Yaskawa INFORM job: long_pipe_cylinder_program.JBI

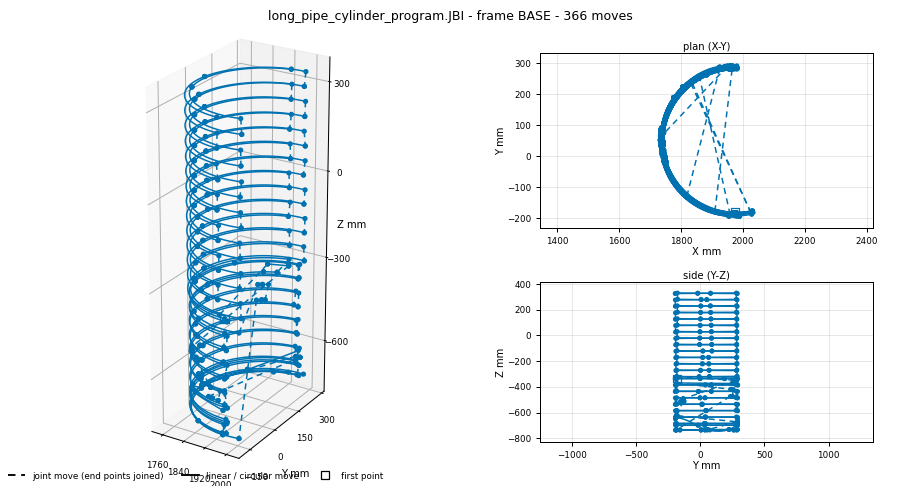
[picture p0: tool path of long_pipe_cylinder_program.JBI in frame BASE, 366 of 497 moves have a stored position in this frame; points joined in program order, loops and branches not executed]
/JOB
//NAME long_pipe_cylinder_program
//POS
///NPOS 488,0,488,0,0,0
///TOOL 0
///POSTYPE BASE
///RECTAN
///RCONF 0,0,0,0,0,0,0,0,0,0,0,0,0,0,0,0,0,0,0,0,0,0,0,0
C00000=1972.508334,-180.722400,-334.797447,175.000000,-89.735184,90.500621
C00001=1972.508334,-180.722400,-334.797447,175.000000,-89.735184,90.500621
C00002=1736.408412,94.560328,-335.864178,175.000000,-89.992940,-9.264169
C00003=1775.133773,190.860038,-336.344108,-5.000000,-89.891094,145.451183
C00004=1775.133773,190.860038,-336.344108,-5.000000,-89.891094,145.451183
C00005=1775.133773,190.860038,-336.344108,-5.000000,-89.891094,145.451183
C00006=1827.250532,245.393825,-336.642454,5.000000,-89.819004,127.146501
C00007=1960.064613,293.278571,-336.981034,-5.000000,-89.737192,92.507006
C00008=1958.169423,292.965805,-385.452719,-5.000000,-89.737685,92.955150
C00009=1958.169423,292.965805,-385.452719,-5.000000,-89.737685,92.955150
C00010=1816.172076,236.277891,-385.065300,-5.000000,-89.831298,130.571443
C00011=1735.474228,88.397981,-384.309626,-175.000000,-89.986107,-7.813258
C00012=1735.474228,88.397981,-384.309626,-175.000000,-89.986107,-7.813258
C00013=1735.474228,88.397981,-384.309626,-175.000000,-89.986107,-7.813258
C00014=1785.900263,-92.792903,-383.515122,175.000000,-89.794130,38.916534
C00015=1972.374520,-180.947584,-383.271088,175.000000,-89.735163,90.478593
C00016=1969.015250,-181.182972,-433.141929,175.000000,-89.734453,89.677478
C00017=1969.015250,-181.182972,-433.141929,175.000000,-89.734453,89.677478
C00018=1788.215870,-95.899703,-433.377664,175.000000,-89.791415,39.815407
C00019=1735.352609,87.595450,-434.180691,175.000000,-89.985451,-7.673859
C00020=1735.352609,87.595450,-434.180691,175.000000,-89.985451,-7.673859
C00021=1735.352609,87.595450,-434.180691,175.000000,-89.985451,-7.673859
C00022=1805.125009,226.010115,-434.882928,-5.000000,-89.844866,134.170721
C00023=1947.373302,291.934457,-435.313330,5.000000,-89.740867,95.560664
C00024=1940.676594,290.957693,-485.903239,5.000000,-89.743112,97.178090
C00025=1940.676594,290.957693,-485.903239,5.000000,-89.743112,97.178090
C00026=1806.475544,227.120060,-485.489579,5.000000,-89.843066,133.702612
C00027=1733.832144,38.186072,-484.550920,-175.000000,-89.930125,5.000000
C00028=1733.832144,38.186072,-484.550920,-175.000000,-89.930125,5.000000
C00029=1733.832144,38.186072,-484.550920,-175.000000,-89.930125,5.000000
C00030=1801.988125,-111.319855,-483.918715,175.000000,-89.777364,44.777879
C00031=1967.484314,-181.404185,-483.739882,-175.000000,-89.734152,89.318297
C00032=1979.401274,-181.476259,-533.747056,175.000000,-89.736874,92.209028
C00033=1979.401274,-181.476259,-533.747056,175.000000,-89.736874,92.209028
C00034=1821.064603,-128.831806,-533.851447,175.000000,-89.762098,51.008369
C00035=1736.221976,17.364408,-534.453644,175.000000,-89.907608,9.246629
C00036=1736.221976,17.364408,-534.453644,175.000000,-89.907608,9.246629
C00037=1736.221976,17.364408,-534.453644,175.000000,-89.907608,9.246629
C00038=1787.842464,206.956552,-535.376849,5.000000,-89.869317,140.291943
C00039=1956.911466,292.208440,-535.920338,5.000000,-89.737992,93.227517
C00040=1950.680326,291.548047,-585.654124,5.000000,-89.739789,94.726243
C00041=1950.680326,291.548047,-585.654124,5.000000,-89.739789,94.726243
C00042=1792.775612,212.526390,-585.149306,5.000000,-89.861770,138.445142
C00043=1733.319404,44.964590,-584.321201,175.000000,-89.938134,5.000000
C00044=1733.319404,44.964590,-584.321201,175.000000,-89.938134,5.000000
C00045=1733.319404,44.964590,-584.321201,175.000000,-89.938134,5.000000
C00046=1826.635210,-133.468869,-583.577209,-175.000000,-89.758362,52.733042
C00047=1971.739744,-181.877826,-583.480783,175.000000,-89.735062,90.367778
C00048=1971.702534,-182.110717,-633.797386,-175.000000,-89.735064,90.369485
C00049=1971.702534,-182.110717,-633.797386,-175.000000,-89.735064,90.369485
C00050=1827.055515,-134.054392,-633.892582,175.000000,-89.758066,52.873969
C00051=1733.473975,40.872659,-634.620107,175.000000,-89.933859,5.000000
C00052=1733.473975,40.872659,-634.620107,175.000000,-89.933859,5.000000
C00053=1733.473975,40.872659,-634.620107,175.000000,-89.933859,5.000000
C00054=1792.290752,211.795028,-635.463207,-5.000000,-89.862421,138.605884
C00055=1947.450954,291.030161,-635.966599,5.000000,-89.740785,95.498948
C00056=1950.402769,291.069729,-685.572290,5.000000,-89.739847,94.772222
C00057=1950.402769,291.069729,-685.572290,5.000000,-89.739847,94.772222
C00058=1804.325673,224.287077,-685.134545,5.000000,-89.845621,134.366136
C00059=1733.942614,33.751843,-684.190461,175.000000,-89.926259,5.086090
C00060=1733.942614,33.751843,-684.190461,175.000000,-89.926259,5.086090
C00061=1733.942614,33.751843,-684.190461,175.000000,-89.926259,5.086090
C00062=1831.125071,-137.328437,-683.483916,175.000000,-89.755535,54.110506
C00063=1976.553212,-182.258277,-683.403882,-175.000000,-89.736196,91.552306
C00064=1977.797365,-182.451641,-733.470089,-175.000000,-89.736513,91.863719
C00065=1977.797365,-182.451641,-733.470089,-175.000000,-89.736513,91.863719
C00066=1832.240189,-138.393667,-733.545972,-175.000000,-89.754849,54.455487
C00067=1732.965067,54.885977,-734.353455,175.000000,-89.949963,-5.000000
C00068=1732.965067,54.885977,-734.353455,175.000000,-89.949963,-5.000000
C00069=1732.965067,54.885977,-734.353455,175.000000,-89.949963,-5.000000
C00070=1795.566929,215.069330,-735.150167,5.000000,-89.857527,137.391169
C00071=1959.659103,291.432152,-648.357585,-5.000000,-89.737207,92.520217
C00072=1954.235485,290.902862,-698.306483,-5.000000,-89.738684,93.822137
C00073=1954.235485,290.902862,-698.306483,-5.000000,-89.738684,93.822137
C00074=1797.089158,216.524941,-698.129153,-5.000000,-89.855307,136.834972
C00075=1743.660264,-16.242507,-697.715930,175.000000,-89.872933,17.309849
C00076=1743.660264,-16.242507,-697.715930,175.000000,-89.872933,17.309849
C00077=1743.660264,-16.242507,-697.715930,175.000000,-89.872933,17.309849
C00078=1826.609334,-134.510209,-697.541573,175.000000,-89.758266,52.778835
C00079=1980.284076,-182.588600,-697.509479,175.000000,-89.737158,92.475638
C00080=1963.195867,-182.887095,-735.326535,-175.000000,-89.733394,88.353627
C00081=1963.195867,-182.887095,-735.326535,-175.000000,-89.733394,88.353627
C00082=1816.510486,-126.597836,-735.374855,175.000000,-89.765173,49.658472
C00083=1737.516210,7.512714,-735.577440,-175.000000,-89.898405,11.339291
C00084=1737.516210,7.512714,-735.577440,-175.000000,-89.898405,11.339291
C00085=1737.516210,7.512714,-735.577440,-175.000000,-89.898405,11.339291
C00086=1770.184921,181.794183,-735.884464,5.000000,-89.899679,147.427154
C00087=1925.404749,287.022342,-736.113649,-175.000000,-60.000000,-79.157724
C00088=1954.714747,-193.319715,326.566406,5.000000,-89.456000,-93.567339
C00089=1954.714747,-193.319715,326.566406,5.000000,-89.456000,-93.567339
C00090=1779.619946,-99.163395,327.312391,-5.000000,-89.635698,-142.973579
C00091=1734.628999,81.575451,328.985260,175.000000,-89.961340,-9.072278
C00092=1734.628999,81.575451,328.985260,175.000000,-89.961340,-9.072278
C00093=1734.628999,81.575451,328.985260,175.000000,-89.961340,-9.072278
C00094=1817.345576,226.880631,330.428549,-175.000000,-89.613678,-50.226634
C00095=1980.685637,281.657087,331.081997,-175.000000,-89.456271,-92.692092
C00096=1975.331224,282.321864,281.169566,-175.000000,-89.456908,-91.391494
C00097=1975.331224,282.321864,281.169566,-175.000000,-89.456908,-91.391494
C00098=1806.653771,217.858300,280.420044,175.000000,-89.637458,-46.774255
C00099=1731.827481,52.492803,278.793480,5.000000,-89.970734,175.000000
C00100=1731.827481,52.492803,278.793480,5.000000,-89.970734,175.000000
C00101=1731.827481,52.492803,278.793480,5.000000,-89.970734,175.000000
C00102=1788.634891,-109.869774,277.304259,5.000000,-89.612008,-139.519963
C00103=1955.354656,-192.883892,276.656769,5.000000,-89.456036,-93.422839
C00104=1953.241860,-192.282365,227.745608,5.000000,-89.455922,-93.942585
C00105=1953.241860,-192.282365,227.745608,5.000000,-89.455922,-93.942585
C00106=1805.749479,-127.416353,228.237298,5.000000,-89.574365,-133.539245
C00107=1734.368459,80.302128,230.143603,175.000000,-89.966442,-8.533915
C00108=1734.368459,80.302128,230.143603,175.000000,-89.966442,-8.533915
C00109=1734.368459,80.302128,230.143603,175.000000,-89.966442,-8.533915
C00110=1827.599341,235.823990,231.692259,175.000000,-89.593399,-53.345559
C00111=1980.201861,282.618326,232.261298,-175.000000,-89.456324,-92.555776
C00112=1977.844791,283.196392,181.219557,175.000000,-89.456586,-91.977383
C00113=1977.844791,283.196392,181.219557,175.000000,-89.456586,-91.977383
C00114=1800.614926,212.840705,180.407208,175.000000,-89.652270,-44.715535
C00115=1734.671921,82.485007,179.119248,175.000000,-89.962516,-8.948170
C00116=1734.671921,82.485007,179.119248,175.000000,-89.962516,-8.948170
C00117=1734.671921,82.485007,179.119248,175.000000,-89.962516,-8.948170
C00118=1775.815306,-92.383268,177.498740,5.000000,-89.647135,-144.574723
C00119=1951.488512,-191.668695,176.704704,-5.000000,-89.455862,-94.376235
C00120=1956.296565,-191.511118,126.598565,5.000000,-89.456090,-93.225427
C00121=1956.296565,-191.511118,126.598565,5.000000,-89.456090,-93.225427
C00122=1767.398896,-79.172346,127.505165,5.000000,-89.674478,-148.258247
C00123=1734.897298,84.109732,129.023199,175.000000,-89.959857,-9.228817
C00124=1734.897298,84.109732,129.023199,175.000000,-89.959857,-9.228817
C00125=1734.897298,84.109732,129.023199,175.000000,-89.959857,-9.228817
C00126=1813.190108,225.089245,130.421898,-175.000000,-89.622936,-48.858885
C00127=1976.049655,283.726966,131.111484,175.000000,-89.456824,-91.534787
C00128=1980.343703,284.039913,81.981880,175.000000,-89.456323,-92.560087
C00129=1980.343703,284.039913,81.981880,175.000000,-89.456323,-92.560087
C00130=1804.393738,217.432812,81.206058,-175.000000,-89.643208,-45.967475
C00131=1735.189988,86.095506,79.906112,-175.000000,-89.956341,-9.600136
C00132=1735.189988,86.095506,79.906112,-175.000000,-89.956341,-9.600136
C00133=1735.189988,86.095506,79.906112,-175.000000,-89.956341,-9.600136
C00134=1760.047671,-65.884409,78.488690,5.000000,-89.702230,-151.824094
C00135=1954.293720,-190.922109,77.466362,5.000000,-89.455966,-93.718563
C00136=1952.261030,-190.301711,27.124546,5.000000,-89.455880,-94.219424
C00137=1952.261030,-190.301711,27.124546,5.000000,-89.455880,-94.219424
C00138=1771.749852,-84.881332,27.972626,-5.000000,-89.660171,-146.354530
C00139=1735.436141,87.763326,29.576092,175.000000,-89.953585,-9.891308
C00140=1735.436141,87.763326,29.576092,175.000000,-89.953585,-9.891308
C00141=1735.436141,87.763326,29.576092,175.000000,-89.953585,-9.891308
C00142=1807.857666,221.152725,30.898117,175.000000,-89.635134,-47.103300
C00143=1980.425383,284.514593,31.640434,175.000000,-89.456319,-92.569770
C00144=1974.499385,285.179775,-18.267395,-175.000000,-89.457069,-91.131550
C00145=1974.499385,285.179775,-18.267395,-175.000000,-89.457069,-91.131550
C00146=1792.515923,205.949239,-19.167650,175.000000,-89.673928,-41.810930
C00147=1735.592913,88.893179,-20.322308,175.000000,-89.952063,-10.052118
C00148=1735.592913,88.893179,-20.322308,175.000000,-89.952063,-10.052118
C00149=1735.592913,88.893179,-20.322308,175.000000,-89.952063,-10.052118
C00150=1768.035641,-78.584750,-21.880090,-5.000000,-89.672697,-148.023907
C00151=1957.112660,-190.135299,-22.779084,-5.000000,-89.456142,-93.058269
C00152=1954.940310,-189.534063,-72.713074,-5.000000,-89.455994,-93.592390
C00153=1954.940310,-189.534063,-72.713074,-5.000000,-89.455994,-93.592390
C00154=1772.096519,-84.332612,-71.868996,5.000000,-89.659321,-146.239795
C00155=1735.849108,90.560889,-70.244197,-175.000000,-89.949296,-10.344614
C00156=1735.849108,90.560889,-70.244197,-175.000000,-89.949296,-10.344614
C00157=1735.849108,90.560889,-70.244197,-175.000000,-89.949296,-10.344614
C00158=1807.335261,221.533864,-68.945810,175.000000,-89.636539,-46.904132
C00159=1980.981190,285.437832,-68.197471,-175.000000,-89.456274,-92.683940
C00160=1976.954500,286.068414,-118.357107,175.000000,-89.456730,-91.703253
C00161=1976.954500,286.068414,-118.357107,175.000000,-89.456730,-91.703253
C00162=1794.437453,208.928718,-119.238021,175.000000,-89.668930,-42.471118
C00163=1736.086800,92.097439,-120.391733,-175.000000,-89.946837,-10.604717
C00164=1736.086800,92.097439,-120.391733,-175.000000,-89.946837,-10.604717
C00165=1736.086800,92.097439,-120.391733,-175.000000,-89.946837,-10.604717
C00166=1770.555957,-81.460267,-122.005364,-5.000000,-89.664470,-146.931728
C00167=1957.534905,-189.205848,-122.870092,-5.000000,-89.456169,-92.976329
C00168=1955.541636,-188.623967,-172.251306,5.000000,-89.456024,-93.467077
C00169=1955.541636,-188.623967,-172.251306,5.000000,-89.456024,-93.467077
C00170=1778.531438,-92.431721,-171.487642,5.000000,-89.639981,-143.577792
C00171=1732.719813,66.430676,-170.022441,5.000000,-89.992920,175.000000
C00172=1732.719813,66.430676,-170.022441,5.000000,-89.992920,175.000000
C00173=1732.719813,66.430676,-170.022441,5.000000,-89.992920,175.000000
C00174=1788.840669,203.012332,-168.683701,-175.000000,-89.684603,-40.419478
C00175=1981.477970,286.360153,-167.735673,175.000000,-89.456236,-92.783945
C00176=1979.440675,286.930016,-218.225518,-175.000000,-89.456441,-92.282657
C00177=1979.440675,286.930016,-218.225518,-175.000000,-89.456441,-92.282657
C00178=1790.115538,204.926497,-219.158085,175.000000,-89.681084,-40.875491
C00179=1732.838504,67.915658,-220.501843,5.000000,-89.995231,175.000000
C00180=1732.838504,67.915658,-220.501843,5.000000,-89.995231,175.000000
C00181=1732.838504,67.915658,-220.501843,5.000000,-89.995231,175.000000
C00182=1789.203829,-105.326756,-222.094371,5.000000,-89.611621,-139.461745
C00183=1953.599312,-188.017562,-222.740726,5.000000,-89.455922,-93.946000
C00184=1951.614652,-187.398418,-272.473730,5.000000,-89.455856,-94.435277
C00185=1951.614652,-187.398418,-272.473730,5.000000,-89.455856,-94.435277
C00186=1767.981489,-75.803835,-271.569815,-5.000000,-89.673597,-148.142414
C00187=1733.025365,70.156398,-270.217707,5.000000,-89.999294,175.000000
C00188=1733.025365,70.156398,-270.217707,5.000000,-89.999294,175.000000
C00189=1733.025365,70.156398,-270.217707,5.000000,-89.999294,175.000000
C00190=1791.376153,206.795190,-268.876581,175.000000,-89.677655,-41.322377
C00191=1977.389681,287.474914,-267.959279,-175.000000,-89.456689,-91.778392
C00192=1980.127143,287.843964,-317.414754,175.000000,-89.456377,-92.428434
C00193=1980.127143,287.843964,-317.414754,175.000000,-89.456377,-92.428434
C00194=1818.134279,233.229535,-318.065555,175.000000,-89.613147,-50.306123
C00195=1733.189757,72.011609,-319.661249,175.000000,-89.997520,-5.259551
C00196=1733.189757,72.011609,-319.661249,175.000000,-89.997520,-5.259551
C00197=1733.189757,72.011609,-319.661249,175.000000,-89.997520,-5.259551
C00198=1836.586331,-146.672080,-321.644810,5.000000,-89.524676,-124.132966
C00199=1957.892088,-187.331721,-321.929136,-5.000000,-89.456185,-92.929779
C00200=1858.376199,260.482372,-347.351524,-175.000000,-89.543653,-61.991286
C00201=1858.376199,260.482372,-347.351524,-175.000000,-89.543653,-61.991286
C00202=1924.143508,283.861537,-347.075892,175.000000,-89.477257,-78.866012
C00203=1924.143508,283.861537,-347.075892,175.000000,-89.477257,-78.866012
C00204=1924.143508,283.861537,-347.075892,175.000000,-89.477257,-78.866012
C00205=1924.143508,283.861537,-347.075892,175.000000,-89.477257,-78.866012
C00206=1924.143508,283.861537,-347.075892,175.000000,-89.477257,-78.866012
C00207=1924.143508,283.861537,-347.075892,175.000000,-89.477257,-78.866012
C00208=1817.788123,-130.782789,-493.061006,-5.000000,-89.553415,-129.847070
C00209=1817.788123,-130.782789,-493.061006,-5.000000,-89.553415,-129.847070
C00210=1817.788123,-130.782789,-493.061006,-5.000000,-89.553415,-129.847070
C00211=1817.788123,-130.782789,-493.061006,-5.000000,-89.553415,-129.847070
C00212=1817.788123,-130.782789,-493.061006,-5.000000,-89.553415,-129.847070
C00213=1817.788123,-130.782789,-493.061006,-5.000000,-89.553415,-129.847070
C00214=1817.788123,-130.782789,-493.061006,-5.000000,-89.553415,-129.847070
C00215=1820.529299,-133.035803,-493.080055,5.000000,-89.548826,-128.992334
C00216=1846.897424,-151.372118,-513.205722,5.000000,-89.511856,-121.226978
C00217=1846.897424,-151.372118,-513.205722,5.000000,-89.511856,-121.226978
C00218=1821.321367,-133.471921,-513.057521,5.000000,-89.547556,-128.752369
C00219=1820.236406,-132.595907,-513.050130,5.000000,-89.549336,-129.088278
C00220=1820.236406,-132.595907,-513.050130,5.000000,-89.549336,-129.088278
C00221=1820.236406,-132.595907,-513.050130,5.000000,-89.549336,-129.088278
C00222=1819.786863,-132.229847,-513.047038,5.000000,-89.550081,-129.227928
C00223=1809.329664,-123.174146,-512.970010,5.000000,-89.568636,-132.560641
C00224=1918.939245,-179.526830,-587.256966,5.000000,-89.460441,-102.462621
C00225=1918.939245,-179.526830,-587.256966,5.000000,-89.460441,-102.462621
C00226=1918.939245,-179.526830,-587.256966,5.000000,-89.460441,-102.462621
C00227=1918.939245,-179.526830,-587.256966,5.000000,-89.460441,-102.462621
C00228=1918.939245,-179.526830,-587.256966,5.000000,-89.460441,-102.462621
C00229=1918.939245,-179.526830,-587.256966,5.000000,-89.460441,-102.462621
C00230=1918.939245,-179.526830,-587.256966,5.000000,-89.460441,-102.462621
C00231=1957.635320,-184.795419,-587.274794,5.000000,-89.456146,-93.044513
C00232=1949.073339,-183.838549,-623.587343,5.000000,-89.455831,-95.119604
C00233=1949.073339,-183.838549,-623.587343,5.000000,-89.455831,-95.119604
C00234=1933.902772,-181.986445,-623.582373,5.000000,-89.457028,-98.801813
C00235=1925.490306,-180.528857,-623.575543,5.000000,-89.458674,-100.858598
C00236=1925.490306,-180.528857,-623.575543,5.000000,-89.458674,-100.858598
C00237=1925.490306,-180.528857,-623.575543,5.000000,-89.458674,-100.858598
C00238=1910.613584,-177.177620,-623.556145,-5.000000,-89.463346,-104.532684
C00239=1908.855039,-176.714605,-623.553220,5.000000,-89.464051,-104.970739
C00240=1965.807687,292.185051,-672.311679,-175.000000,-89.458919,-88.890807
C00241=1965.807687,292.185051,-672.311679,-175.000000,-89.458919,-88.890807
C00242=1965.807687,292.185051,-672.311679,-175.000000,-89.458919,-88.890807
C00243=1965.807687,292.185051,-672.311679,-175.000000,-89.458919,-88.890807
C00244=1965.807687,292.185051,-672.311679,-175.000000,-89.458919,-88.890807
C00245=1965.807687,292.185051,-672.311679,-175.000000,-89.458919,-88.890807
C00246=1965.807687,292.185051,-672.311679,-175.000000,-89.458919,-88.890807
C00247=1949.617497,291.318971,-672.319655,175.000000,-89.464120,-84.984527
C00248=1732.686632,61.358656,-731.853025,5.000000,-89.967260,175.000000
C00249=1732.686632,61.358656,-731.853025,5.000000,-89.967260,175.000000
C00250=1761.922582,169.336891,-731.466710,-175.000000,-89.780816,-28.750237
C00251=1803.937484,224.772179,-731.260128,175.000000,-89.646098,-45.565709
C00252=1803.937484,224.772179,-731.260128,175.000000,-89.646098,-45.565709
C00253=1803.937484,224.772179,-731.260128,175.000000,-89.646098,-45.565709
C00254=1890.457969,278.927524,-731.044422,175.000000,-89.505428,-70.345572
C00255=1979.850375,292.599397,-730.969320,-175.000000,-60.000000,-92.262460
C00256=1988.952084,-193.321978,-335.660245,5.000000,-89.736885,-87.731834
C00257=1988.952084,-193.321978,-335.660245,5.000000,-89.736885,-87.731834
C00258=1922.586515,-186.559330,-335.687073,5.000000,-89.730402,-103.904663
C00259=1746.425890,0.354695,-334.975890,5.000000,-89.902247,-169.489126
C00260=1746.425890,0.354695,-334.975890,5.000000,-89.902247,-169.489126
C00261=1746.425890,0.354695,-334.975890,5.000000,-89.902247,-169.489126
C00262=1787.054580,182.047852,-334.098954,-175.000000,-89.885858,-35.720088
C00263=1962.442340,280.110057,-333.491213,-175.000000,-89.739008,-85.858326
C00264=1962.239094,280.322063,-383.166333,-175.000000,-89.739081,-85.798541
C00265=1962.239094,280.322063,-383.166333,-175.000000,-89.739081,-85.798541
C00266=1807.540169,206.989598,-383.641436,-175.000000,-89.853881,-43.475372
C00267=1742.500791,41.615558,-384.464192,-5.000000,-89.947315,-175.000000
C00268=1742.500791,41.615558,-384.464192,-5.000000,-89.947315,-175.000000
C00269=1742.500791,41.615558,-384.464192,-5.000000,-89.947315,-175.000000
C00270=1821.954194,-133.274193,-385.204421,5.000000,-89.768453,-131.673551
C00271=1988.957882,-193.093466,-385.335105,5.000000,-89.736875,-87.740955
C00272=1985.673220,-192.969637,-435.382757,5.000000,-89.736050,-88.545662
C00273=1985.673220,-192.969637,-435.382757,5.000000,-89.736050,-88.545662
C00274=1838.144346,-146.190690,-435.295395,5.000000,-89.757159,-126.640515
C00275=1749.557100,-13.208123,-434.757222,5.000000,-89.887199,-166.020933
C00276=1749.557100,-13.208123,-434.757222,5.000000,-89.887199,-166.020933
C00277=1749.557100,-13.208123,-434.757222,5.000000,-89.887199,-166.020933
C00278=1786.148374,181.117360,-433.825328,175.000000,-89.887626,-35.306804
C00279=1964.929440,280.733300,-433.207419,-175.000000,-89.738320,-86.439498
C00280=1962.929130,280.829623,-483.398301,175.000000,-89.738905,-85.944438
C00281=1962.929130,280.829623,-483.398301,175.000000,-89.738905,-85.944438
C00282=1799.026883,197.874467,-483.926026,175.000000,-89.866420,-40.364219
C00283=1746.794667,-0.211956,-484.889039,5.000000,-89.900886,-169.179134
C00284=1746.794667,-0.211956,-484.889039,5.000000,-89.900886,-169.179134
C00285=1746.794667,-0.211956,-484.889039,5.000000,-89.900886,-169.179134
C00286=1830.599752,-140.071935,-485.463247,5.000000,-89.762139,-128.961304
C00287=1988.334115,-192.656369,-485.568551,5.000000,-89.736694,-87.913019
C00288=1978.718558,-192.579897,-535.575683,-5.000000,-89.734476,-90.247506
C00289=1978.718558,-192.579897,-535.575683,-5.000000,-89.734476,-90.247506
C00290=1829.485888,-138.898248,-535.457850,5.000000,-89.762948,-129.321970
C00291=1744.723341,13.039165,-534.828555,5.000000,-89.915006,-172.366737
C00292=1744.723341,13.039165,-534.828555,5.000000,-89.915006,-172.366737
C00293=1744.723341,13.039165,-534.828555,5.000000,-89.915006,-172.366737
C00294=1801.344355,200.741406,-533.909782,175.000000,-89.862990,-41.205269
C00295=1956.432208,280.506326,-533.404552,175.000000,-89.740910,-84.358255
C00296=1960.714239,281.116737,-583.095370,175.000000,-89.739587,-85.386546
C00297=1960.714239,281.116737,-583.095370,175.000000,-89.739587,-85.386546
C00298=1798.943757,198.135301,-583.621349,175.000000,-89.866681,-40.300580
C00299=1742.684968,47.807133,-584.366741,-5.000000,-89.953209,175.000000
C00300=1742.684968,47.807133,-584.366741,-5.000000,-89.953209,175.000000
C00301=1742.684968,47.807133,-584.366741,-5.000000,-89.953209,175.000000
C00302=1826.002318,-135.721463,-585.143588,5.000000,-89.765499,-130.432538
C00303=1979.551635,-192.351895,-585.271294,5.000000,-89.734641,-90.056725
C00304=1987.992632,-191.978943,-635.494749,-5.000000,-89.736575,-88.027341
C00305=1987.992632,-191.978943,-635.494749,-5.000000,-89.736575,-88.027341
C00306=1828.203070,-137.304478,-635.381567,-5.000000,-89.763924,-129.751320
C00307=1742.729939,41.885794,-634.626699,-5.000000,-89.946324,-175.000000
C00308=1742.729939,41.885794,-634.626699,-5.000000,-89.946324,-175.000000
C00309=1742.729939,41.885794,-634.626699,-5.000000,-89.946324,-175.000000
C00310=1797.387591,196.460896,-633.863043,-175.000000,-89.869153,-39.699058
C00311=1968.836143,281.862517,-633.317379,175.000000,-89.737303,-87.342467
C00312=1954.664260,281.004839,-683.259671,-175.000000,-89.741531,-83.896917
C00313=1954.664260,281.004839,-683.259671,-175.000000,-89.741531,-83.896917
C00314=1795.584014,194.438901,-683.799891,-175.000000,-89.872065,-38.995027
C00315=1742.836095,38.962696,-684.566046,-5.000000,-89.942808,-175.000000
C00316=1742.836095,38.962696,-684.566046,-5.000000,-89.942808,-175.000000
C00317=1742.836095,38.962696,-684.566046,-5.000000,-89.942808,-175.000000
C00318=1824.163425,-133.598262,-685.293850,5.000000,-89.766947,-131.046960
C00319=1988.135684,-191.744342,-685.419442,5.000000,-89.736600,-88.003328
C00320=1972.052967,-191.526506,-648.429379,5.000000,-89.733171,-91.900839
C00321=1972.052967,-191.526506,-648.429379,5.000000,-89.733171,-91.900839
C00322=1827.103536,-135.847991,-648.381311,5.000000,-89.764784,-130.125242
C00323=1742.933944,37.414856,-734.871085,5.000000,-89.940827,-175.000000
C00324=1742.933944,37.414856,-734.871085,5.000000,-89.940827,-175.000000
C00325=1742.933944,37.414856,-734.871085,5.000000,-89.940827,-175.000000
C00326=1793.521685,192.031976,-734.110801,175.000000,-89.875465,-38.178983
C00327=1961.465151,281.862500,-733.547699,-175.000000,-89.739401,-85.536614
C00328=1967.741442,282.497863,-697.257401,175.000000,-89.737630,-87.045893
C00329=1967.741442,282.497863,-697.257401,175.000000,-89.737630,-87.045893
C00330=1792.835573,191.329737,-697.468805,-175.000000,-89.876662,-37.892977
C00331=1743.066273,35.352986,-697.750192,-5.000000,-89.938282,-175.000000
C00332=1743.066273,35.352986,-697.750192,-5.000000,-89.938282,-175.000000
C00333=1743.066273,35.352986,-697.750192,-5.000000,-89.938282,-175.000000
C00334=1822.129897,-131.268027,-698.008217,5.000000,-89.768589,-131.729833
C00335=1975.447994,-191.384219,-698.061141,-5.000000,-89.733783,-91.090715
C00336=1970.460702,-191.059856,-735.980414,-5.000000,-89.732886,-92.304386
C00337=1970.460702,-191.059856,-735.980414,-5.000000,-89.732886,-92.304386
C00338=1774.497667,164.178247,-735.439120,-175.000000,-89.911127,-29.930092
C00339=1882.583601,262.056095,-735.237808,175.000000,-89.778732,-65.744304
C00340=1882.583601,262.056095,-735.237808,175.000000,-89.778732,-65.744304
C00341=1882.583601,262.056095,-735.237808,175.000000,-89.778732,-65.744304
C00342=1935.146540,278.708726,-735.192558,-175.000000,-89.748973,-79.097537
C00343=1967.804699,282.674977,-735.175298,180.000000,-60.000000,-87.053161
C00344=1923.594334,288.562657,326.309286,5.000000,-89.456493,103.394594
C00345=1923.594334,288.562657,326.309286,5.000000,-89.456493,103.394594
C00346=1778.931380,186.296279,327.012165,5.000000,-89.625807,147.123951
C00347=1753.174038,-18.438247,328.878865,-175.000000,-89.924540,18.537239
C00348=1753.174038,-18.438247,328.878865,-175.000000,-89.924540,18.537239
C00349=1753.174038,-18.438247,328.878865,-175.000000,-89.924540,18.537239
C00350=1845.989241,-140.212091,330.177497,175.000000,-89.611724,56.087847
C00351=2027.210017,-175.666758,330.824163,-175.000000,-89.455950,101.769696
C00352=2030.458035,-175.444910,281.624416,175.000000,-89.456156,102.548916
C00353=2030.458035,-175.444910,281.624416,175.000000,-89.456156,102.548916
C00354=1850.410526,-143.517777,281.012730,175.000000,-89.603503,57.337154
C00355=1746.009327,7.776774,279.418290,175.000000,-89.987574,11.875009
C00356=1746.009327,7.776774,279.418290,175.000000,-89.987574,11.875009
C00357=1746.009327,7.776774,279.418290,175.000000,-89.987574,11.875009
C00358=1797.499225,210.710489,277.613222,5.000000,-89.577618,139.653999
C00359=1926.435953,288.742116,277.109227,5.000000,-89.456212,102.713145
C00360=1924.517191,287.813766,227.139871,5.000000,-89.456409,103.208997
C00361=1924.517191,287.813766,227.139871,5.000000,-89.456409,103.208997
C00362=1802.431768,215.771986,227.599873,5.000000,-89.567218,137.883161
C00363=1746.537824,5.256565,229.468059,175.000000,-89.982771,12.380956
C00364=1746.537824,5.256565,229.468059,175.000000,-89.982771,12.380956
C00365=1746.537824,5.256565,229.468059,175.000000,-89.982771,12.380956
C00366=1874.012665,-157.238470,231.207263,-175.000000,-89.563828,63.842875
C00367=2027.457608,-176.577374,231.655082,-175.000000,-89.455954,101.788035
C00368=2028.556050,-176.835513,181.191493,-175.000000,-89.456009,102.036782
C00369=2028.556050,-176.835513,181.191493,-175.000000,-89.456009,102.036782
C00370=1855.284942,-147.391288,180.614792,175.000000,-89.594929,58.671859
C00371=1746.761464,4.171553,179.010667,175.000000,-89.981333,12.532355
C00372=1746.761464,4.171553,179.010667,175.000000,-89.981333,12.532355
C00373=1746.761464,4.171553,179.010667,175.000000,-89.981333,12.532355
C00374=1796.535107,208.421163,177.190324,5.000000,-89.580179,140.079788
C00375=1926.162717,287.702513,176.675864,-5.000000,-89.456252,102.823925
C00376=1921.535318,286.109795,126.481424,-5.000000,-89.456802,103.991565
C00377=1921.535318,286.109795,126.481424,-5.000000,-89.456802,103.991565
C00378=1799.123372,210.891931,126.970511,5.000000,-89.574617,139.150122
C00379=1747.107563,2.553313,128.825128,-175.000000,-89.978640,12.816148
C00380=1747.107563,2.553313,128.825128,-175.000000,-89.978640,12.816148
C00381=1747.107563,2.553313,128.825128,-175.000000,-89.978640,12.816148
C00382=1858.583232,-149.779742,130.441586,175.000000,-89.589265,59.572974
C00383=2030.641106,-176.869420,130.994190,175.000000,-89.456149,102.529224
C00384=2026.326438,-178.266913,81.416811,175.000000,-89.455894,101.445370
C00385=2026.326438,-178.266913,81.416811,175.000000,-89.455894,101.445370
C00386=1858.422891,-150.097588,80.861362,175.000000,-89.589695,59.503988
C00387=1747.653374,0.110531,79.265974,175.000000,-89.973995,13.305698
C00388=1747.653374,0.110531,79.265974,175.000000,-89.973995,13.305698
C00389=1747.653374,0.110531,79.265974,175.000000,-89.973995,13.305698
C00390=1775.795062,178.266467,77.651585,5.000000,-89.637130,148.744432
C00391=1923.659425,286.144939,76.901883,5.000000,-89.456536,103.486272
C00392=1925.746012,286.147013,26.764517,-5.000000,-89.456317,102.991561
C00393=1925.746012,286.147013,26.764517,-5.000000,-89.456317,102.991561
C00394=1789.039491,197.240613,27.356514,5.000000,-89.598922,143.087181
C00395=1747.882879,-0.954727,29.135339,175.000000,-89.972592,13.453521
C00396=1747.882879,-0.954727,29.135339,175.000000,-89.972592,13.453521
C00397=1747.882879,-0.954727,29.135339,175.000000,-89.972592,13.453521
C00398=1856.847600,-149.577494,30.712782,-175.000000,-89.592615,59.038033
C00399=2028.089189,-178.389701,31.280047,175.000000,-89.455968,101.857414
C00400=2030.482536,-178.354482,-18.098128,-175.000000,-89.456116,102.425909
C00401=2030.482536,-178.354482,-18.098128,-175.000000,-89.456116,102.425909
C00402=1855.487950,-149.164298,-18.675459,175.000000,-89.595188,58.631024
C00403=1748.335112,-2.924302,-20.227499,-175.000000,-89.969046,13.827418
C00404=1748.335112,-2.924302,-20.227499,-175.000000,-89.969046,13.827418
C00405=1748.335112,-2.924302,-20.227499,-175.000000,-89.969046,13.827418
C00406=1779.910718,183.608902,-21.914124,-5.000000,-89.624678,146.959945
C00407=1921.237583,284.577663,-22.610698,5.000000,-89.456882,104.130114
C00408=1923.447554,284.632491,-72.838786,5.000000,-89.456594,103.603520
C00409=1923.447554,284.632491,-72.838786,5.000000,-89.456594,103.603520
C00410=1794.947065,203.639696,-72.306383,5.000000,-89.584843,140.845448
C00411=1748.687099,-4.456752,-70.444003,175.000000,-89.966544,14.091358
C00412=1748.687099,-4.456752,-70.444003,175.000000,-89.966544,14.091358
C00413=1748.687099,-4.456752,-70.444003,175.000000,-89.966544,14.091358
C00414=1842.588785,-141.123116,-69.004430,175.000000,-89.619777,54.890181
C00415=2026.057204,-179.772155,-68.324025,-175.000000,-89.455876,101.315002
C00416=2028.112746,-179.834927,-118.149333,-175.000000,-89.455956,101.799031
C00417=2028.112746,-179.834927,-118.149333,-175.000000,-89.455956,101.799031
C00418=1838.246501,-138.398122,-118.866910,175.000000,-89.628811,53.575261
C00419=1743.680129,21.725396,-120.526655,-5.000000,-89.971388,-172.447245
C00420=1743.680129,21.725396,-120.526655,-5.000000,-89.971388,-172.447245
C00421=1743.680129,21.725396,-120.526655,-5.000000,-89.971388,-172.447245
C00422=1797.243004,205.846979,-122.152468,-5.000000,-89.579759,140.010207
C00423=1926.767153,284.925577,-122.665215,-5.000000,-89.456245,102.803656
C00424=1921.265264,283.116276,-172.759557,5.000000,-89.456917,104.188335
C00425=1921.265264,283.116276,-172.759557,5.000000,-89.456917,104.188335
C00426=1806.556787,215.747594,-172.330338,5.000000,-89.560310,136.666434
C00427=1743.847455,20.660700,-170.618075,5.000000,-89.972764,-172.302198
C00428=1743.847455,20.660700,-170.618075,5.000000,-89.972764,-172.302198
C00429=1743.847455,20.660700,-170.618075,5.000000,-89.972764,-172.302198
C00430=1838.610555,-139.069792,-168.961657,175.000000,-89.628237,53.658028
C00431=2030.237101,-179.867981,-168.246977,-175.000000,-89.456079,102.300764
C00432=2025.902472,-181.254125,-218.132279,175.000000,-89.455865,101.212783
C00433=2025.902472,-181.254125,-218.132279,175.000000,-89.455865,101.212783
C00434=1842.596985,-142.343931,-218.814838,-175.000000,-89.620285,54.815581
C00435=1744.185616,18.389165,-220.486972,-5.000000,-89.976930,-171.863070
C00436=1744.185616,18.389165,-220.486972,-5.000000,-89.976930,-171.863070
C00437=1744.185616,18.389165,-220.486972,-5.000000,-89.976930,-171.863070
C00438=1792.324432,198.627841,-222.085978,5.000000,-89.591759,141.959023
C00439=1925.293807,283.611168,-222.647855,-5.000000,-89.456409,103.211056
C00440=1927.311993,283.584763,-273.085155,-5.000000,-89.456219,102.733919
C00441=1927.311993,283.584763,-273.085155,-5.000000,-89.456219,102.733919
C00442=1791.582947,197.090527,-272.513976,5.000000,-89.593809,142.284445
C00443=1746.839787,3.259330,-270.782146,175.000000,-89.989025,11.722215
C00444=1746.839787,3.259330,-270.782146,175.000000,-89.989025,11.722215
C00445=1746.839787,3.259330,-270.782146,175.000000,-89.989025,11.722215
C00446=1847.016517,-145.797326,-269.215958,175.000000,-89.611760,56.082407
C00447=2029.932704,-180.908941,-268.569543,175.000000,-89.456046,102.182576
C00448=2031.954700,-180.949736,-318.566126,-175.000000,-89.456193,102.659810
C00449=2031.954700,-180.949736,-318.566126,-175.000000,-89.456193,102.659810
C00450=1865.543351,-157.482096,-319.075077,175.000000,-89.578793,61.283405
C00451=1749.403048,-7.895058,-320.674021,-175.000000,-89.963950,14.365026
C00452=1749.403048,-7.895058,-320.674021,-175.000000,-89.963950,14.365026
C00453=1749.403048,-7.895058,-320.674021,-175.000000,-89.963950,14.365026
C00454=1799.486078,206.204274,-322.585790,5.000000,-89.575540,139.305713
C00455=1926.030136,282.804203,-323.080585,-5.000000,-89.456350,103.072267
C00456=1888.640150,270.287588,-373.403349,-5.000000,-89.467720,112.566067
C00457=1888.640150,270.287588,-373.403349,-5.000000,-89.467720,112.566067
C00458=1854.452380,252.717920,-373.298850,-5.000000,-89.492892,121.835532
C00459=1849.344538,249.455874,-373.277289,-5.000000,-89.498086,123.295504
C00460=1849.344538,249.455874,-373.277289,-5.000000,-89.498086,123.295504
C00461=1849.344538,249.455874,-373.277289,-5.000000,-89.498086,123.295504
C00462=1832.907960,237.630608,-373.195507,-5.000000,-89.517786,128.174584
C00463=2025.513614,-182.790804,-368.934661,175.000000,-89.455850,101.052703
C00464=1834.806442,238.625141,-418.367227,5.000000,-89.515364,127.619121
C00465=1834.806442,238.625141,-418.367227,5.000000,-89.515364,127.619121
C00466=1846.163008,246.854292,-418.424281,5.000000,-89.501621,124.240259
C00467=1846.926572,247.371793,-418.427783,-5.000000,-89.500777,124.018062
C00468=1846.926572,247.371793,-418.427783,-5.000000,-89.500777,124.018062
C00469=1846.926572,247.371793,-418.427783,-5.000000,-89.500777,124.018062
C00470=1850.158251,249.514784,-418.442163,5.000000,-89.497313,123.083970
C00471=1863.665147,257.688537,-418.494954,5.000000,-89.484596,119.280227
C00472=1854.758695,251.859361,-473.914585,-5.000000,-89.492765,121.798473
C00473=1854.758695,251.859361,-473.914585,-5.000000,-89.492765,121.798473
C00474=1846.640605,246.595043,-473.879572,5.000000,-89.501199,124.129367
C00475=1845.276543,245.663621,-473.873252,5.000000,-89.502721,124.527250
C00476=1845.276543,245.663621,-473.873252,5.000000,-89.502721,124.527250
C00477=1845.276543,245.663621,-473.873252,5.000000,-89.502721,124.527250
C00478=1842.516698,243.736123,-473.860062,5.000000,-89.505899,125.338161
C00479=1831.374035,235.334287,-473.801023,-5.000000,-89.520121,128.700304
C00480=2027.732910,-186.725528,-734.776427,175.000000,-89.455888,101.404113
C00481=2027.732910,-186.725528,-734.776427,175.000000,-89.455888,101.404113
C00482=1953.504754,-189.861860,-734.813362,-175.000000,-89.479975,83.434276
C00483=1855.460190,-155.780460,-734.993968,175.000000,-89.597756,58.228098
C00484=1855.460190,-155.780460,-734.993968,175.000000,-89.597756,58.228098
C00485=1855.460190,-155.780460,-734.993968,175.000000,-89.597756,58.228098
C00486=1765.336581,-54.536811,-735.401110,-175.000000,-89.863264,25.119101
C00487=1744.625372,75.511105,-735.862945,-175.000000,-60.000000,-7.021335
///POSTYPE PULSE
///PULSE
EX00000=70656.0
EX00001=132096.0
EX00002=254976.0
EX00003=332800.0
///POSTYPE PULSE
///PULSE
EC00000=70656.0
EC00001=70656.0
EC00002=70656.0
EC00003=70656.0
EC00004=70656.0
EC00005=70656.0
EC00006=70656.0
EC00007=70656.0
EC00008=70656.0
EC00009=70656.0
EC00010=70656.0
EC00011=70656.0
EC00012=70656.0
EC00013=70656.0
EC00014=70656.0
EC00015=70656.0
EC00016=70656.0
EC00017=70656.0
EC00018=70656.0
EC00019=70656.0
EC00020=70656.0
EC00021=70656.0
EC00022=70656.0
EC00023=70656.0
EC00024=70656.0
EC00025=70656.0
EC00026=70656.0
EC00027=70656.0
EC00028=70656.0
EC00029=70656.0
EC00030=70656.0
EC00031=70656.0
EC00032=70656.0
EC00033=70656.0
EC00034=70656.0
EC00035=70656.0
EC00036=70656.0
EC00037=70656.0
EC00038=70656.0
EC00039=70656.0
EC00040=70656.0
EC00041=70656.0
EC00042=70656.0
EC00043=70656.0
EC00044=70656.0
EC00045=70656.0
EC00046=70656.0
EC00047=70656.0
EC00048=70656.0
EC00049=70656.0
EC00050=70656.0
EC00051=70656.0
EC00052=70656.0
EC00053=70656.0
EC00054=70656.0
EC00055=70656.0
EC00056=70656.0
EC00057=70656.0
EC00058=70656.0
EC00059=70656.0
EC00060=70656.0
EC00061=70656.0
EC00062=70656.0
EC00063=70656.0
EC00064=70656.0
EC00065=70656.0
EC00066=70656.0
EC00067=70656.0
EC00068=70656.0
EC00069=70656.0
EC00070=70656.0
EC00071=70656.0
EC00072=70656.0
EC00073=70656.0
EC00074=70656.0
EC00075=70656.0
EC00076=70656.0
EC00077=70656.0
EC00078=70656.0
EC00079=70656.0
EC00080=70656.0
EC00081=70656.0
EC00082=70656.0
EC00083=70656.0
EC00084=70656.0
EC00085=70656.0
EC00086=70656.0
EC00087=70656.0
EC00088=132096.0
EC00089=132096.0
EC00090=132096.0
EC00091=132096.0
EC00092=132096.0
EC00093=132096.0
EC00094=132096.0
EC00095=132096.0
EC00096=132096.0
EC00097=132096.0
EC00098=132096.0
EC00099=132096.0
EC00100=132096.0
EC00101=132096.0
EC00102=132096.0
EC00103=132096.0
EC00104=132096.0
EC00105=132096.0
EC00106=132096.0
EC00107=132096.0
EC00108=132096.0
EC00109=132096.0
EC00110=132096.0
EC00111=132096.0
EC00112=132096.0
EC00113=132096.0
EC00114=132096.0
EC00115=132096.0
EC00116=132096.0
EC00117=132096.0
EC00118=132096.0
EC00119=132096.0
EC00120=132096.0
EC00121=132096.0
EC00122=132096.0
EC00123=132096.0
EC00124=132096.0
EC00125=132096.0
EC00126=132096.0
EC00127=132096.0
EC00128=132096.0
EC00129=132096.0
EC00130=132096.0
EC00131=132096.0
EC00132=132096.0
EC00133=132096.0
EC00134=132096.0
EC00135=132096.0
EC00136=132096.0
EC00137=132096.0
EC00138=132096.0
EC00139=132096.0
EC00140=132096.0
EC00141=132096.0
EC00142=132096.0
EC00143=132096.0
EC00144=132096.0
EC00145=132096.0
EC00146=132096.0
EC00147=132096.0
EC00148=132096.0
EC00149=132096.0
EC00150=132096.0
EC00151=132096.0
EC00152=132096.0
EC00153=132096.0
EC00154=132096.0
EC00155=132096.0
EC00156=132096.0
EC00157=132096.0
EC00158=132096.0
EC00159=132096.0
EC00160=132096.0
EC00161=132096.0
EC00162=132096.0
EC00163=132096.0
EC00164=132096.0
EC00165=132096.0
EC00166=132096.0
EC00167=132096.0
EC00168=132096.0
EC00169=132096.0
EC00170=132096.0
EC00171=132096.0
EC00172=132096.0
EC00173=132096.0
EC00174=132096.0
EC00175=132096.0
EC00176=132096.0
EC00177=132096.0
EC00178=132096.0
EC00179=132096.0
EC00180=132096.0
EC00181=132096.0
EC00182=132096.0
EC00183=132096.0
EC00184=132096.0
EC00185=132096.0
EC00186=132096.0
EC00187=132096.0
EC00188=132096.0
EC00189=132096.0
EC00190=132096.0
EC00191=132096.0
EC00192=132096.0
EC00193=132096.0
EC00194=132096.0
EC00195=132096.0
EC00196=132096.0
EC00197=132096.0
EC00198=132096.0
EC00199=132096.0
EC00200=132096.0
EC00201=132096.0
EC00202=132096.0
EC00203=132096.0
EC00204=132096.0
EC00205=132096.0
EC00206=132096.0
EC00207=132096.0
EC00208=132096.0
EC00209=132096.0
EC00210=132096.0
EC00211=132096.0
EC00212=132096.0
EC00213=132096.0
EC00214=132096.0
EC00215=132096.0
EC00216=132096.0
EC00217=132096.0
EC00218=132096.0
EC00219=132096.0
EC00220=132096.0
EC00221=132096.0
EC00222=132096.0
EC00223=132096.0
EC00224=132096.0
EC00225=132096.0
EC00226=132096.0
EC00227=132096.0
EC00228=132096.0
EC00229=132096.0
EC00230=132096.0
EC00231=132096.0
EC00232=132096.0
EC00233=132096.0
EC00234=132096.0
EC00235=132096.0
EC00236=132096.0
EC00237=132096.0
EC00238=132096.0
EC00239=132096.0
EC00240=132096.0
EC00241=132096.0
EC00242=132096.0
EC00243=132096.0
EC00244=132096.0
EC00245=132096.0
EC00246=132096.0
EC00247=132096.0
EC00248=132096.0
EC00249=132096.0
EC00250=132096.0
EC00251=132096.0
EC00252=132096.0
EC00253=132096.0
EC00254=132096.0
EC00255=132096.0
EC00256=254976.0
EC00257=254976.0
EC00258=254976.0
EC00259=254976.0
EC00260=254976.0
EC00261=254976.0
EC00262=254976.0
EC00263=254976.0
EC00264=254976.0
EC00265=254976.0
EC00266=254976.0
EC00267=254976.0
EC00268=254976.0
EC00269=254976.0
EC00270=254976.0
EC00271=254976.0
EC00272=254976.0
EC00273=254976.0
EC00274=254976.0
EC00275=254976.0
EC00276=254976.0
EC00277=254976.0
EC00278=254976.0
EC00279=254976.0
EC00280=254976.0
EC00281=254976.0
EC00282=254976.0
EC00283=254976.0
EC00284=254976.0
EC00285=254976.0
EC00286=254976.0
EC00287=254976.0
EC00288=254976.0
EC00289=254976.0
EC00290=254976.0
EC00291=254976.0
EC00292=254976.0
EC00293=254976.0
EC00294=254976.0
EC00295=254976.0
EC00296=254976.0
EC00297=254976.0
EC00298=254976.0
EC00299=254976.0
EC00300=254976.0
EC00301=254976.0
EC00302=254976.0
EC00303=254976.0
EC00304=254976.0
EC00305=254976.0
EC00306=254976.0
EC00307=254976.0
EC00308=254976.0
EC00309=254976.0
EC00310=254976.0
EC00311=254976.0
EC00312=254976.0
EC00313=254976.0
EC00314=254976.0
EC00315=254976.0
EC00316=254976.0
EC00317=254976.0
EC00318=254976.0
EC00319=254976.0
EC00320=254976.0
EC00321=254976.0
EC00322=254976.0
EC00323=254976.0
EC00324=254976.0
EC00325=254976.0
EC00326=254976.0
EC00327=254976.0
EC00328=254976.0
EC00329=254976.0
EC00330=254976.0
EC00331=254976.0
EC00332=254976.0
EC00333=254976.0
EC00334=254976.0
EC00335=254976.0
EC00336=254976.0
EC00337=254976.0
EC00338=254976.0
EC00339=254976.0
EC00340=254976.0
EC00341=254976.0
EC00342=254976.0
EC00343=254976.0
EC00344=332800.0
EC00345=332800.0
EC00346=332800.0
EC00347=332800.0
EC00348=332800.0
EC00349=332800.0
EC00350=332800.0
EC00351=332800.0
EC00352=332800.0
EC00353=332800.0
EC00354=332800.0
EC00355=332800.0
EC00356=332800.0
EC00357=332800.0
EC00358=332800.0
EC00359=332800.0
EC00360=332800.0
EC00361=332800.0
EC00362=332800.0
EC00363=332800.0
EC00364=332800.0
EC00365=332800.0
EC00366=332800.0
EC00367=332800.0
EC00368=332800.0
EC00369=332800.0
EC00370=332800.0
EC00371=332800.0
EC00372=332800.0
EC00373=332800.0
EC00374=332800.0
EC00375=332800.0
EC00376=332800.0
EC00377=332800.0
EC00378=332800.0
EC00379=332800.0
EC00380=332800.0
EC00381=332800.0
EC00382=332800.0
EC00383=332800.0
EC00384=332800.0
EC00385=332800.0
EC00386=332800.0
EC00387=332800.0
EC00388=332800.0
EC00389=332800.0
EC00390=332800.0
EC00391=332800.0
EC00392=332800.0
EC00393=332800.0
EC00394=332800.0
EC00395=332800.0
EC00396=332800.0
EC00397=332800.0
EC00398=332800.0
EC00399=332800.0
EC00400=332800.0
EC00401=332800.0
EC00402=332800.0
EC00403=332800.0
EC00404=332800.0
EC00405=332800.0
EC00406=332800.0
EC00407=332800.0
EC00408=332800.0
EC00409=332800.0
EC00410=332800.0
EC00411=332800.0
EC00412=332800.0
EC00413=332800.0
EC00414=332800.0
EC00415=332800.0
EC00416=332800.0
EC00417=332800.0
EC00418=332800.0
EC00419=332800.0
EC00420=332800.0
EC00421=332800.0
EC00422=332800.0
EC00423=332800.0
EC00424=332800.0
EC00425=332800.0
EC00426=332800.0
EC00427=332800.0
EC00428=332800.0
EC00429=332800.0
EC00430=332800.0
EC00431=332800.0
EC00432=332800.0
EC00433=332800.0
EC00434=332800.0
EC00435=332800.0
EC00436=332800.0
EC00437=332800.0
EC00438=332800.0
EC00439=332800.0
EC00440=332800.0
EC00441=332800.0
EC00442=332800.0
EC00443=332800.0
EC00444=332800.0
EC00445=332800.0
EC00446=332800.0
EC00447=332800.0
EC00448=332800.0
EC00449=332800.0
EC00450=332800.0
EC00451=332800.0
EC00452=332800.0
EC00453=332800.0
EC00454=332800.0
EC00455=332800.0
EC00456=332800.0
EC00457=332800.0
EC00458=332800.0
EC00459=332800.0
EC00460=332800.0
EC00461=332800.0
EC00462=332800.0
EC00463=332800.0
EC00464=332800.0
EC00465=332800.0
EC00466=332800.0
EC00467=332800.0
EC00468=332800.0
EC00469=332800.0
EC00470=332800.0
EC00471=332800.0
EC00472=332800.0
EC00473=332800.0
EC00474=332800.0
EC00475=332800.0
EC00476=332800.0
EC00477=332800.0
EC00478=332800.0
EC00479=332800.0
EC00480=332800.0
EC00481=332800.0
EC00482=332800.0
EC00483=332800.0
EC00484=332800.0
EC00485=332800.0
EC00486=332800.0
EC00487=332800.0
//INST
///DATE 2023/08/13 14:29
///ATTR SC,RW,RJ
////FRAME BASE
///GROUP1 RB1,ST1
NOP
MOVJ P009 EX000 VJ=15.00
MOVJ C00000 EC00000 VJ=15.0
CALL JOB:SPYON
MOVC C00001 EC00001 V=150.0
MOVC C00002 EC00002 V=150.0
MOVC C00003 EC00003 V=150.0
MOVJ C00004 EC00004 VJ=15.0
MOVC C00005 EC00005 V=150.0
MOVC C00006 EC00006 V=150.0
MOVC C00007 EC00007 V=150.0
MOVJ C00008 EC00008 VJ=15.0
MOVC C00009 EC00009 V=150.0
MOVC C00010 EC00010 V=150.0
MOVC C00011 EC00011 V=150.0
MOVJ C00012 EC00012 VJ=15.0
MOVC C00013 EC00013 V=150.0
MOVC C00014 EC00014 V=150.0
MOVC C00015 EC00015 V=150.0
MOVJ C00016 EC00016 VJ=15.0
MOVC C00017 EC00017 V=150.0
MOVC C00018 EC00018 V=150.0
MOVC C00019 EC00019 V=150.0
MOVJ C00020 EC00020 VJ=15.0
MOVC C00021 EC00021 V=150.0
MOVC C00022 EC00022 V=150.0
MOVC C00023 EC00023 V=150.0
MOVJ C00024 EC00024 VJ=15.0
MOVC C00025 EC00025 V=150.0
MOVC C00026 EC00026 V=150.0
MOVC C00027 EC00027 V=150.0
MOVJ C00028 EC00028 VJ=15.0
MOVC C00029 EC00029 V=150.0
MOVC C00030 EC00030 V=150.0
MOVC C00031 EC00031 V=150.0
MOVJ C00032 EC00032 VJ=15.0
MOVC C00033 EC00033 V=150.0
MOVC C00034 EC00034 V=150.0
MOVC C00035 EC00035 V=150.0
MOVJ C00036 EC00036 VJ=15.0
MOVC C00037 EC00037 V=150.0
MOVC C00038 EC00038 V=150.0
MOVC C00039 EC00039 V=150.0
MOVJ C00040 EC00040 VJ=15.0
MOVC C00041 EC00041 V=150.0
MOVC C00042 EC00042 V=150.0
MOVC C00043 EC00043 V=150.0
MOVJ C00044 EC00044 VJ=15.0
MOVC C00045 EC00045 V=150.0
MOVC C00046 EC00046 V=150.0
MOVC C00047 EC00047 V=150.0
MOVJ C00048 EC00048 VJ=15.0
MOVC C00049 EC00049 V=150.0
MOVC C00050 EC00050 V=150.0
MOVC C00051 EC00051 V=150.0
MOVJ C00052 EC00052 VJ=15.0
MOVC C00053 EC00053 V=150.0
MOVC C00054 EC00054 V=150.0
MOVC C00055 EC00055 V=150.0
MOVJ C00056 EC00056 VJ=15.0
MOVC C00057 EC00057 V=150.0
MOVC C00058 EC00058 V=150.0
MOVC C00059 EC00059 V=150.0
MOVJ C00060 EC00060 VJ=15.0
MOVC C00061 EC00061 V=150.0
MOVC C00062 EC00062 V=150.0
MOVC C00063 EC00063 V=150.0
MOVJ C00064 EC00064 VJ=15.0
MOVC C00065 EC00065 V=150.0
MOVC C00066 EC00066 V=150.0
MOVC C00067 EC00067 V=150.0
MOVJ C00068 EC00068 VJ=15.0
MOVC C00069 EC00069 V=150.0
MOVC C00070 EC00070 V=150.0
MOVC C00071 EC00071 V=150.0
MOVJ C00072 EC00072 VJ=15.0
MOVC C00073 EC00073 V=150.0
MOVC C00074 EC00074 V=150.0
MOVC C00075 EC00075 V=150.0
MOVJ C00076 EC00076 VJ=15.0
MOVC C00077 EC00077 V=150.0
MOVC C00078 EC00078 V=150.0
MOVC C00079 EC00079 V=150.0
MOVJ C00080 EC00080 VJ=15.0
MOVC C00081 EC00081 V=150.0
MOVC C00082 EC00082 V=150.0
MOVC C00083 EC00083 V=150.0
MOVJ C00084 EC00084 VJ=15.0
MOVC C00085 EC00085 V=150.0
MOVC C00086 EC00086 V=150.0
MOVC C00087 EC00087 V=150.0
CALL JOB:SPYOF
MOVJ P009 VJ=15.00
MOVL P009 EX00000 V=150.0
MOVJ C00088 EC00088 VJ=15.0
CALL JOB:SPYON
MOVC C00089 EC00089 V=150.0
MOVC C00090 EC00090 V=150.0
MOVC C00091 EC00091 V=150.0
MOVJ C00092 EC00092 VJ=15.0
MOVC C00093 EC00093 V=150.0
MOVC C00094 EC00094 V=150.0
MOVC C00095 EC00095 V=150.0
MOVJ C00096 EC00096 VJ=15.0
MOVC C00097 EC00097 V=150.0
MOVC C00098 EC00098 V=150.0
MOVC C00099 EC00099 V=150.0
MOVJ C00100 EC00100 VJ=15.0
MOVC C00101 EC00101 V=150.0
MOVC C00102 EC00102 V=150.0
MOVC C00103 EC00103 V=150.0
MOVJ C00104 EC00104 VJ=15.0
MOVC C00105 EC00105 V=150.0
MOVC C00106 EC00106 V=150.0
MOVC C00107 EC00107 V=150.0
MOVJ C00108 EC00108 VJ=15.0
MOVC C00109 EC00109 V=150.0
MOVC C00110 EC00110 V=150.0
MOVC C00111 EC00111 V=150.0
MOVJ C00112 EC00112 VJ=15.0
MOVC C00113 EC00113 V=150.0
MOVC C00114 EC00114 V=150.0
MOVC C00115 EC00115 V=150.0
MOVJ C00116 EC00116 VJ=15.0
MOVC C00117 EC00117 V=150.0
MOVC C00118 EC00118 V=150.0
MOVC C00119 EC00119 V=150.0
MOVJ C00120 EC00120 VJ=15.0
MOVC C00121 EC00121 V=150.0
MOVC C00122 EC00122 V=150.0
MOVC C00123 EC00123 V=150.0
MOVJ C00124 EC00124 VJ=15.0
MOVC C00125 EC00125 V=150.0
MOVC C00126 EC00126 V=150.0
MOVC C00127 EC00127 V=150.0
MOVJ C00128 EC00128 VJ=15.0
MOVC C00129 EC00129 V=150.0
MOVC C00130 EC00130 V=150.0
MOVC C00131 EC00131 V=150.0
MOVJ C00132 EC00132 VJ=15.0
MOVC C00133 EC00133 V=150.0
MOVC C00134 EC00134 V=150.0
MOVC C00135 EC00135 V=150.0
MOVJ C00136 EC00136 VJ=15.0
MOVC C00137 EC00137 V=150.0
MOVC C00138 EC00138 V=150.0
MOVC C00139 EC00139 V=150.0
MOVJ C00140 EC00140 VJ=15.0
MOVC C00141 EC00141 V=150.0
MOVC C00142 EC00142 V=150.0
MOVC C00143 EC00143 V=150.0
MOVJ C00144 EC00144 VJ=15.0
MOVC C00145 EC00145 V=150.0
MOVC C00146 EC00146 V=150.0
MOVC C00147 EC00147 V=150.0
MOVJ C00148 EC00148 VJ=15.0
MOVC C00149 EC00149 V=150.0
MOVC C00150 EC00150 V=150.0
MOVC C00151 EC00151 V=150.0
MOVJ C00152 EC00152 VJ=15.0
MOVC C00153 EC00153 V=150.0
MOVC C00154 EC00154 V=150.0
MOVC C00155 EC00155 V=150.0
MOVJ C00156 EC00156 VJ=15.0
MOVC C00157 EC00157 V=150.0
MOVC C00158 EC00158 V=150.0
MOVC C00159 EC00159 V=150.0
MOVJ C00160 EC00160 VJ=15.0
MOVC C00161 EC00161 V=150.0
MOVC C00162 EC00162 V=150.0
MOVC C00163 EC00163 V=150.0
MOVJ C00164 EC00164 VJ=15.0
MOVC C00165 EC00165 V=150.0
MOVC C00166 EC00166 V=150.0
MOVC C00167 EC00167 V=150.0
MOVJ C00168 EC00168 VJ=15.0
MOVC C00169 EC00169 V=150.0
MOVC C00170 EC00170 V=150.0
MOVC C00171 EC00171 V=150.0
MOVJ C00172 EC00172 VJ=15.0
MOVC C00173 EC00173 V=150.0
MOVC C00174 EC00174 V=150.0
MOVC C00175 EC00175 V=150.0
MOVJ C00176 EC00176 VJ=15.0
MOVC C00177 EC00177 V=150.0
MOVC C00178 EC00178 V=150.0
MOVC C00179 EC00179 V=150.0
MOVJ C00180 EC00180 VJ=15.0
MOVC C00181 EC00181 V=150.0
MOVC C00182 EC00182 V=150.0
MOVC C00183 EC00183 V=150.0
MOVJ C00184 EC00184 VJ=15.0
MOVC C00185 EC00185 V=150.0
MOVC C00186 EC00186 V=150.0
MOVC C00187 EC00187 V=150.0
MOVJ C00188 EC00188 VJ=15.0
MOVC C00189 EC00189 V=150.0
MOVC C00190 EC00190 V=150.0
MOVC C00191 EC00191 V=150.0
MOVJ C00192 EC00192 VJ=15.0
MOVC C00193 EC00193 V=150.0
MOVC C00194 EC00194 V=150.0
MOVC C00195 EC00195 V=150.0
MOVJ C00196 EC00196 VJ=15.0
MOVC C00197 EC00197 V=150.0
MOVC C00198 EC00198 V=150.0
MOVC C00199 EC00199 V=150.0
MOVJ C00200 EC00200 VJ=15.0
MOVC C00201 EC00201 V=150.0
MOVC C00202 EC00202 V=150.0
MOVC C00203 EC00203 V=150.0
MOVJ C00204 EC00204 VJ=15.0
MOVC C00205 EC00205 V=150.0
MOVC C00206 EC00206 V=150.0
MOVC C00207 EC00207 V=150.0
MOVJ C00208 EC00208 VJ=15.0
MOVC C00209 EC00209 V=150.0
MOVC C00210 EC00210 V=150.0
MOVC C00211 EC00211 V=150.0
MOVJ C00212 EC00212 VJ=15.0
MOVC C00213 EC00213 V=150.0
MOVC C00214 EC00214 V=150.0
MOVC C00215 EC00215 V=150.0
MOVJ C00216 EC00216 VJ=15.0
MOVC C00217 EC00217 V=150.0
MOVC C00218 EC00218 V=150.0
MOVC C00219 EC00219 V=150.0
MOVJ C00220 EC00220 VJ=15.0
MOVC C00221 EC00221 V=150.0
MOVC C00222 EC00222 V=150.0
MOVC C00223 EC00223 V=150.0
MOVJ C00224 EC00224 VJ=15.0
MOVC C00225 EC00225 V=150.0
MOVC C00226 EC00226 V=150.0
MOVC C00227 EC00227 V=150.0
MOVJ C00228 EC00228 VJ=15.0
MOVC C00229 EC00229 V=150.0
MOVC C00230 EC00230 V=150.0
MOVC C00231 EC00231 V=150.0
MOVJ C00232 EC00232 VJ=15.0
MOVC C00233 EC00233 V=150.0
MOVC C00234 EC00234 V=150.0
MOVC C00235 EC00235 V=150.0
MOVJ C00236 EC00236 VJ=15.0
MOVC C00237 EC00237 V=150.0
MOVC C00238 EC00238 V=150.0
MOVC C00239 EC00239 V=150.0
MOVJ C00240 EC00240 VJ=15.0
MOVC C00241 EC00241 V=150.0
MOVC C00242 EC00242 V=150.0
MOVC C00243 EC00243 V=150.0
MOVJ C00244 EC00244 VJ=15.0
MOVC C00245 EC00245 V=150.0
MOVC C00246 EC00246 V=150.0
MOVC C00247 EC00247 V=150.0
MOVJ C00248 EC00248 VJ=15.0
MOVC C00249 EC00249 V=150.0
MOVC C00250 EC00250 V=150.0
MOVC C00251 EC00251 V=150.0
MOVJ C00252 EC00252 VJ=15.0
MOVC C00253 EC00253 V=150.0
MOVC C00254 EC00254 V=150.0
MOVC C00255 EC00255 V=150.0
CALL JOB:SPYOF
MOVJ P009 VJ=15.00
MOVL P009 EX00001 V=150.0
MOVJ C00256 EC00256 VJ=15.0
CALL JOB:SPYON
MOVC C00257 EC00257 V=150.0
MOVC C00258 EC00258 V=150.0
MOVC C00259 EC00259 V=150.0
MOVJ C00260 EC00260 VJ=15.0
MOVC C00261 EC00261 V=150.0
MOVC C00262 EC00262 V=150.0
MOVC C00263 EC00263 V=150.0
MOVJ C00264 EC00264 VJ=15.0
MOVC C00265 EC00265 V=150.0
MOVC C00266 EC00266 V=150.0
MOVC C00267 EC00267 V=150.0
MOVJ C00268 EC00268 VJ=15.0
MOVC C00269 EC00269 V=150.0
MOVC C00270 EC00270 V=150.0
MOVC C00271 EC00271 V=150.0
MOVJ C00272 EC00272 VJ=15.0
MOVC C00273 EC00273 V=150.0
MOVC C00274 EC00274 V=150.0
MOVC C00275 EC00275 V=150.0
MOVJ C00276 EC00276 VJ=15.0
MOVC C00277 EC00277 V=150.0
MOVC C00278 EC00278 V=150.0
MOVC C00279 EC00279 V=150.0
MOVJ C00280 EC00280 VJ=15.0
MOVC C00281 EC00281 V=150.0
MOVC C00282 EC00282 V=150.0
MOVC C00283 EC00283 V=150.0
MOVJ C00284 EC00284 VJ=15.0
MOVC C00285 EC00285 V=150.0
MOVC C00286 EC00286 V=150.0
MOVC C00287 EC00287 V=150.0
MOVJ C00288 EC00288 VJ=15.0
MOVC C00289 EC00289 V=150.0
MOVC C00290 EC00290 V=150.0
MOVC C00291 EC00291 V=150.0
MOVJ C00292 EC00292 VJ=15.0
MOVC C00293 EC00293 V=150.0
MOVC C00294 EC00294 V=150.0
MOVC C00295 EC00295 V=150.0
MOVJ C00296 EC00296 VJ=15.0
MOVC C00297 EC00297 V=150.0
MOVC C00298 EC00298 V=150.0
MOVC C00299 EC00299 V=150.0
MOVJ C00300 EC00300 VJ=15.0
MOVC C00301 EC00301 V=150.0
MOVC C00302 EC00302 V=150.0
MOVC C00303 EC00303 V=150.0
MOVJ C00304 EC00304 VJ=15.0
MOVC C00305 EC00305 V=150.0
MOVC C00306 EC00306 V=150.0
MOVC C00307 EC00307 V=150.0
MOVJ C00308 EC00308 VJ=15.0
MOVC C00309 EC00309 V=150.0
MOVC C00310 EC00310 V=150.0
MOVC C00311 EC00311 V=150.0
MOVJ C00312 EC00312 VJ=15.0
MOVC C00313 EC00313 V=150.0
MOVC C00314 EC00314 V=150.0
MOVC C00315 EC00315 V=150.0
MOVJ C00316 EC00316 VJ=15.0
MOVC C00317 EC00317 V=150.0
MOVC C00318 EC00318 V=150.0
MOVC C00319 EC00319 V=150.0
MOVJ C00320 EC00320 VJ=15.0
MOVC C00321 EC00321 V=150.0
MOVC C00322 EC00322 V=150.0
MOVC C00323 EC00323 V=150.0
MOVJ C00324 EC00324 VJ=15.0
MOVC C00325 EC00325 V=150.0
MOVC C00326 EC00326 V=150.0
MOVC C00327 EC00327 V=150.0
MOVJ C00328 EC00328 VJ=15.0
MOVC C00329 EC00329 V=150.0
MOVC C00330 EC00330 V=150.0
MOVC C00331 EC00331 V=150.0
MOVJ C00332 EC00332 VJ=15.0
MOVC C00333 EC00333 V=150.0
MOVC C00334 EC00334 V=150.0
MOVC C00335 EC00335 V=150.0
MOVJ C00336 EC00336 VJ=15.0
MOVC C00337 EC00337 V=150.0
MOVC C00338 EC00338 V=150.0
MOVC C00339 EC00339 V=150.0
MOVJ C00340 EC00340 VJ=15.0
MOVC C00341 EC00341 V=150.0
MOVC C00342 EC00342 V=150.0
MOVC C00343 EC00343 V=150.0
CALL JOB:SPYOF
MOVJ P009 VJ=15.00
MOVL P009 EX00002 V=150.0
MOVJ C00344 EC00344 VJ=15.0
CALL JOB:SPYON
MOVC C00345 EC00345 V=150.0
MOVC C00346 EC00346 V=150.0
MOVC C00347 EC00347 V=150.0
MOVJ C00348 EC00348 VJ=15.0
MOVC C00349 EC00349 V=150.0
MOVC C00350 EC00350 V=150.0
MOVC C00351 EC00351 V=150.0
MOVJ C00352 EC00352 VJ=15.0
MOVC C00353 EC00353 V=150.0
MOVC C00354 EC00354 V=150.0
MOVC C00355 EC00355 V=150.0
MOVJ C00356 EC00356 VJ=15.0
MOVC C00357 EC00357 V=150.0
MOVC C00358 EC00358 V=150.0
MOVC C00359 EC00359 V=150.0
MOVJ C00360 EC00360 VJ=15.0
MOVC C00361 EC00361 V=150.0
MOVC C00362 EC00362 V=150.0
MOVC C00363 EC00363 V=150.0
MOVJ C00364 EC00364 VJ=15.0
MOVC C00365 EC00365 V=150.0
MOVC C00366 EC00366 V=150.0
MOVC C00367 EC00367 V=150.0
MOVJ C00368 EC00368 VJ=15.0
MOVC C00369 EC00369 V=150.0
MOVC C00370 EC00370 V=150.0
MOVC C00371 EC00371 V=150.0
MOVJ C00372 EC00372 VJ=15.0
MOVC C00373 EC00373 V=150.0
MOVC C00374 EC00374 V=150.0
MOVC C00375 EC00375 V=150.0
MOVJ C00376 EC00376 VJ=15.0
MOVC C00377 EC00377 V=150.0
MOVC C00378 EC00378 V=150.0
MOVC C00379 EC00379 V=150.0
MOVJ C00380 EC00380 VJ=15.0
MOVC C00381 EC00381 V=150.0
MOVC C00382 EC00382 V=150.0
MOVC C00383 EC00383 V=150.0
MOVJ C00384 EC00384 VJ=15.0
MOVC C00385 EC00385 V=150.0
MOVC C00386 EC00386 V=150.0
MOVC C00387 EC00387 V=150.0
MOVJ C00388 EC00388 VJ=15.0
MOVC C00389 EC00389 V=150.0
MOVC C00390 EC00390 V=150.0
MOVC C00391 EC00391 V=150.0
MOVJ C00392 EC00392 VJ=15.0
MOVC C00393 EC00393 V=150.0
MOVC C00394 EC00394 V=150.0
MOVC C00395 EC00395 V=150.0
MOVJ C00396 EC00396 VJ=15.0
MOVC C00397 EC00397 V=150.0
MOVC C00398 EC00398 V=150.0
MOVC C00399 EC00399 V=150.0
MOVJ C00400 EC00400 VJ=15.0
MOVC C00401 EC00401 V=150.0
MOVC C00402 EC00402 V=150.0
MOVC C00403 EC00403 V=150.0
MOVJ C00404 EC00404 VJ=15.0
MOVC C00405 EC00405 V=150.0
MOVC C00406 EC00406 V=150.0
MOVC C00407 EC00407 V=150.0
MOVJ C00408 EC00408 VJ=15.0
MOVC C00409 EC00409 V=150.0
MOVC C00410 EC00410 V=150.0
MOVC C00411 EC00411 V=150.0
MOVJ C00412 EC00412 VJ=15.0
MOVC C00413 EC00413 V=150.0
MOVC C00414 EC00414 V=150.0
MOVC C00415 EC00415 V=150.0
MOVJ C00416 EC00416 VJ=15.0
MOVC C00417 EC00417 V=150.0
MOVC C00418 EC00418 V=150.0
MOVC C00419 EC00419 V=150.0
MOVJ C00420 EC00420 VJ=15.0
MOVC C00421 EC00421 V=150.0
MOVC C00422 EC00422 V=150.0
MOVC C00423 EC00423 V=150.0
MOVJ C00424 EC00424 VJ=15.0
MOVC C00425 EC00425 V=150.0
MOVC C00426 EC00426 V=150.0
MOVC C00427 EC00427 V=150.0
MOVJ C00428 EC00428 VJ=15.0
MOVC C00429 EC00429 V=150.0
MOVC C00430 EC00430 V=150.0
MOVC C00431 EC00431 V=150.0
MOVJ C00432 EC00432 VJ=15.0
MOVC C00433 EC00433 V=150.0
MOVC C00434 EC00434 V=150.0
MOVC C00435 EC00435 V=150.0
MOVJ C00436 EC00436 VJ=15.0
MOVC C00437 EC00437 V=150.0
MOVC C00438 EC00438 V=150.0
MOVC C00439 EC00439 V=150.0
MOVJ C00440 EC00440 VJ=15.0
MOVC C00441 EC00441 V=150.0
MOVC C00442 EC00442 V=150.0
MOVC C00443 EC00443 V=150.0
MOVJ C00444 EC00444 VJ=15.0
MOVC C00445 EC00445 V=150.0
MOVC C00446 EC00446 V=150.0
MOVC C00447 EC00447 V=150.0
MOVJ C00448 EC00448 VJ=15.0
MOVC C00449 EC00449 V=150.0
MOVC C00450 EC00450 V=150.0
MOVC C00451 EC00451 V=150.0
MOVJ C00452 EC00452 VJ=15.0
MOVC C00453 EC00453 V=150.0
MOVC C00454 EC00454 V=150.0
MOVC C00455 EC00455 V=150.0
MOVJ C00456 EC00456 VJ=15.0
MOVC C00457 EC00457 V=150.0
MOVC C00458 EC00458 V=150.0
MOVC C00459 EC00459 V=150.0
MOVJ C00460 EC00460 VJ=15.0
MOVC C00461 EC00461 V=150.0
MOVC C00462 EC00462 V=150.0
MOVC C00463 EC00463 V=150.0
MOVJ C00464 EC00464 VJ=15.0
MOVC C00465 EC00465 V=150.0
MOVC C00466 EC00466 V=150.0
MOVC C00467 EC00467 V=150.0
MOVJ C00468 EC00468 VJ=15.0
MOVC C00469 EC00469 V=150.0
MOVC C00470 EC00470 V=150.0
MOVC C00471 EC00471 V=150.0
MOVJ C00472 EC00472 VJ=15.0
MOVC C00473 EC00473 V=150.0
MOVC C00474 EC00474 V=150.0
MOVC C00475 EC00475 V=150.0
MOVJ C00476 EC00476 VJ=15.0
MOVC C00477 EC00477 V=150.0
MOVC C00478 EC00478 V=150.0
MOVC C00479 EC00479 V=150.0
MOVJ C00480 EC00480 VJ=15.0
MOVC C00481 EC00481 V=150.0
MOVC C00482 EC00482 V=150.0
MOVC C00483 EC00483 V=150.0
MOVJ C00484 EC00484 VJ=15.0
MOVC C00485 EC00485 V=150.0
MOVC C00486 EC00486 V=150.0
MOVC C00487 EC00487 V=150.0
CALL JOB:SPYOF
MOVJ P009 VJ=15.00
MOVL P009 EX00003 V=150.0
END
